// PROCESS THIS MACHINE CYCLE AS A TIME STEP

FUNCTION RunTime

VAR
	
	// Read in values for easy access
	cycle : REAL := status.time_cycle;
	next  : REAL := status.time_now + userin.time_step;
	cip   : REAL := cycle - status.time_cip;
	
END_VAR

// Loop back to 0 if new time is over
IF next > cycle THEN
	next := 0;
END_IF

// Update CIP status based on the new time
SetCIP(next >= cip);

// Save new time
status.time_now := next;

END_FUNCTION

(* stored: Version 1.1.0.1, ProductVersion 3.1.4024.12
   POU RunTime: Id {32785608-3767-47f1-a28c-91f917ff1a3b}, SpecialFunc None *)
